TYPE ST_FLAGS :
STRUCT
    eDiagnosisType : E_DIAGNOSISTYPE;
    eTimeStampType : E_TIMESTAMPTYPE;
    nNumberOfParametersInDiagnosisMessage : USINT;
END_STRUCT
END_TYPE

(* stored: Version 1.1.0.1
   DUT ST_FLAGS: Id {a22c0de0-4aa7-4870-8fcb-0380fc972d78} *)
